PROGRAM P16_CoverOperation
VAR
// 	isCoverClosed 	: BOOL;

	bCoverCP	: BOOL;
	bLowerLimit	: BOOL;
	bUpperLimit	: BOOL;
	TimerUpLED 		: TON;
	TimerUpLED_X 	: TON;
	TimerDownLED 	: TON;
	TimerDownLED_X 	: TON;
	TimerDownDelayOff 	: TON;
	(* Input *)
	bUpSwitch	: BOOL;
	bDownSwitch 	: BOOL;
	bClamp_Lock_switch: BOOL;
	bClamp_Release_switch: BOOL;
	(* Output *)
	bUpLED 		: BOOL;
	bDownLED 	: BOOL;
	bOnUpRelay 	: BOOL;
	bOnDownRelay : BOOL;
	bOnClamp_Lock_Relay:BOOL;
	bOnClamp_Release_Relay:BOOL;		
	
	bClampLock: BOOL;
	bClampRelease: BOOL;
END_VAR

_DigitalInput();

TimerDownDelayOff(IN:=bLowerLimit, PT:=T#500MS);

//Cover Open 조건
//공정 중이지 않을것
//Dor Pressure down
//Clamp Releaae
//Susceptor down
//CDG 700 torr 이상
//모든 벨브 ff

// Cover Operation Condition
IF P90_Interlock.bReactorOpenEnable THEN
	(*Cover*)
	IF bClampRelease THEN
		bOnUpRelay := (bDownSwitch = FALSE AND bUpSwitch = TRUE AND bUpperLimit = FALSE );
		bOnDownRelay := (bDownSwitch = TRUE AND bUpSwitch = FALSE AND (bLowerLimit = FALSE OR TimerDownDelayOff.Q = FALSE ));
	ELSE
		bOnUpRelay:=FALSE;
		bOnDownRelay:=FALSE;
	END_IF
	(*clamp*)
	bOnClamp_Lock_Relay:=(bClamp_Lock_switch = TRUE AND bClamp_Release_switch = FALSE);
	bOnClamp_Release_Relay:=(bClamp_Lock_switch = FALSE AND bClamp_Release_switch = TRUE);
ELSE
	(*Cover*)
	bOnUpRelay:=FALSE;
	bOnDownRelay:=FALSE;
	(*clamp*)
	bOnClamp_Lock_Relay:=FALSE;
	bOnClamp_Release_Relay:=FALSE;
END_IF

//LED Blinking
TimerUpLED(IN:=(bOnUpRelay AND TimerUpLED_X.Q = FALSE), PT:=T#500MS);
TimerUpLED_X(IN:=TimerUpLED.Q, PT:=T#300MS);
bUpLED := (TimerUpLED.Q AND bOnUpRelay) OR bUpperLimit;

TimerDownLED(IN:=(bOnDownRelay AND TimerDownLED_X.Q = FALSE), PT:=T#500MS);
TimerDownLED_X(IN:=TimerDownLED.Q, PT:=T#300MS);
bDownLED := (TimerDownLED.Q AND bOnDownRelay) OR bLowerLimit;

_DigitalOutput();

ACTION _DigitalInput:
//(* Read from Device Value *)
//// Cover Operation Switch

bUpSwitch 		:=GVL_IO_REACTOR_CABINET.DI_01_ReactorDoorUpButton;
bDownSwitch 	:=GVL_IO_REACTOR_CABINET.DI_01_ReactorDoorDownButton;
bUpperLimit 	:=GVL_IO_REACTOR_CABINET.DI_02_ReactorDoorUpLimitSensor;
bLowerLimit 	:=GVL_IO_REACTOR_CABINET.DI_03_ReactorDoorDownLimitSensor;
bCoverCP 		:= GVL_IO_GAS_CABINET.DI_02_CoverLiftMotorCP;

bClampLock := GVL_IO_REACTOR_CABINET.DI_03_CylinderAutoSwitch_Closed;
bClampRelease :=GVL_IO_REACTOR_CABINET.DI_03_CylinderAutoSwitch_Opened;

bClamp_Lock_switch:=GVL_IO_REACTOR_CABINET.DI_01_ClampLock;
bClamp_Release_switch:=GVL_IO_REACTOR_CABINET.DI_01_ClampRelease;
END_ACTION

ACTION _DigitalOutput:
(* Write to Device Value *)
// Cover Operation Switch Lamp


//Status Output
GVL_IO.isCoverClosed := bLowerLimit;

GVL_IO_REACTOR_CABINET.DO_06_ReactorCoverUpButtonLamp := bUpLED;
GVL_IO_REACTOR_CABINET.DO_06_ReactorCoverDownButtonLamp := bDownLED;

GVL_IO_REACTOR_CABINET.DO_04_ReactorCoverUpRelay :=bOnUpRelay;
GVL_IO_REACTOR_CABINET.DO_04_ReactorCoverDownRelay :=bOnDownRelay;

GVL_IO_REACTOR_CABINET.DO_06_ClampLockButtonLamp := GVL_IO_REACTOR_CABINET.DI_03_CylinderAutoSwitch_Closed;
GVL_IO_REACTOR_CABINET.DO_06_ClampReleaseButtonLamp := GVL_IO_REACTOR_CABINET.DI_03_CylinderAutoSwitch_Opened;

GVL_IO_REACTOR_CABINET.DO_05_ClampLock := bOnClamp_Lock_Relay;
GVL_IO_REACTOR_CABINET.DO_05_ClampRelease := bOnClamp_Release_Relay;
END_ACTION

END_PROGRAM

(* stored: Version 1.1.0.1, ProductVersion 3.1.4024.12
   POU P16_CoverOperation: Id {413bd09a-4287-4ca5-a610-3ab16d733b75}, SpecialFunc None
   Action _DigitalInput: Id {3993b22d-b9e7-4b2a-8103-fff9e7c1039b}
   Action _DigitalOutput: Id {d459d509-027a-4d88-87ff-6244ba761c3e} *)
